// TIA Portal project "Encoder 2" (V16)

(* hardware
DEVICE "S7-1200 station_1"  S7-1200 Station
   slot 0: "Rack_0"  S7-1200 Rack  Rack  V1.0
   slot 1: "Encoder"  CPU 1212C DC/DC/DC  6ES7 212-1AE40-0XB0  V4.3
*)

// ===== PLC "Encoder"  CPU 1212C DC/DC/DC =====

VAR_GLOBAL   // PLC tag table "Default tag table"
   "RESET_ENCODER" AT %I1.0 : Bool;
   "Tag_1" AT %I1.1 : Bool;
   "ENCODER" AT %ID1000 : DWord;
   "Tag_2" AT %MW300 : Int;
   "Tag_3" AT %I0.0 : Bool;
   "Tag_4" AT %Q0.0 : Bool;
END_VAR

ORGANIZATION_BLOCK "Main"   // OB1, LAD, ProgramCycle
TITLE = "Main Program Sweep (Cycle)"
{ S7_Optimized_Access := 'TRUE' }
VERSION : 0.1
   VAR_INPUT
      Initial_Call : Bool;   // Initial call of this OB
      Remanence : Bool;   // =True, if remanent data are available
   END_VAR
BEGIN

REGION Network 1
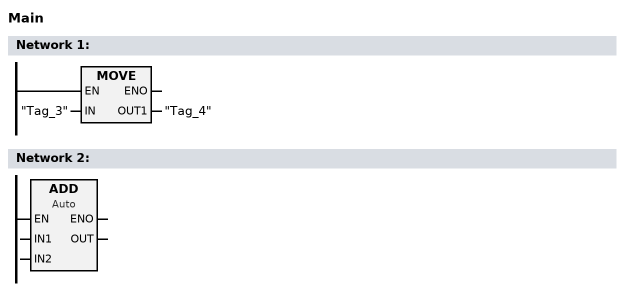
   RUNG wire#powerrail
      Move(in := "Tag_3", out1 => "Tag_4")
   END_RUNG
   // the same network as SCL:
   "Tag_4" := "Tag_3";
END_REGION

REGION Network 2
   RUNG wire#powerrail
      Add(in1 :=, in2 :=, out =>)
   END_RUNG
   // the same network as SCL:
   // no SCL statement known for Add: written as a call
   Add();
END_REGION
END_ORGANIZATION_BLOCK